PROGRAM PRG_DIAGNOSTIC
VAR
   heartbeat AT %Q* : UINT := 0;
END_VAR

heartbeat := heartbeat + 1;
IF heartbeat > 65000
   THEN heartbeat := 0;
END_IF

END_PROGRAM

(* stored: Version 1.1.0.1, ProductVersion 3.1.4022.12
   POU PRG_DIAGNOSTIC: Id {76865f8d-e607-4817-9ebc-004a709e1429}, SpecialFunc None *)
